TYPE ST_Switch :
STRUCT
	bGreenSwitch		:BIT;
	bYellowSwitch		:BIT;
	bRedSwitch			:BIT;
	bWhiteSwitch		:BIT;
	bBlueSwitch			:BIT;
END_STRUCT
END_TYPE

(* stored: Version 1.1.0.1
   DUT ST_Switch: Id {201d54a7-de96-4043-ad13-56fa4d337081} *)
